FUNCTION_BLOCK TM3BC_Ethe_yYhtt9jWKUOJs (* Composite Function Block Type *)
  (* Standard: 61499-2 *)
  (* Version 0.0, 4/12/2022, Schneider Electric, template *)
  PACKAGE Main;
  {SET_ATTRIBUTE(Signature, 9B-51-86-C6-44-F1-B9-23-4E-CE-E4-D3-BB-FD-BE-0A-D2-5B-5E-A3-24-21-0B-6D-81-3C-00-8F-1B-F1-B9-BB-43-CA-DC-29-26-A0-D3-07-47-84-6D-56-70-09-2E-2C-30-58-B0-D9-37-4B-26-3D-BF-E3-73-7B-3A-E4-6A-55_67-4B-EE-2B-F7-15-C2-07-6B-CD-FB-3F-4A-FB-6C-FA-FE-85-84-91-EA-8A-10-A4-3E-5F-A5-D7-87-43-15-4E-8E-61-10-AD-23-0C-80-F7-8B-ED-9D-C9-E2-50-D4-40-3E-AD-16-B1-1E-C7-18-6C-9F-7C-EF-80-0E-8A-1D-44)}
  {SET_ATTRIBUTE(CreationMethod, Generic)}
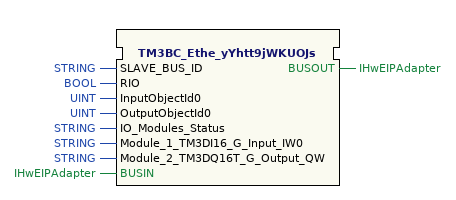
  VAR_INPUT
    SLAVE_BUS_ID : STRING; {SET_ATTRIBUTE(Configuration.HWConfiguration.HideInHwConfigurator, False)} {SET_ATTRIBUTE(Configuration.HWConfiguration.InheritInstanceName, True)}
    RIO : BOOL; {SET_ATTRIBUTE(Configuration.HWConfiguration.HideInHwConfigurator, True)} {SET_ATTRIBUTE(Configuration.HWConfiguration.ReadOnlyInHwConfigurator, True)}
    InputObjectId0 : UINT; (* Object ID of Input connection 0 *) {SET_ATTRIBUTE(Configuration.HWConfiguration.ReadOnlyInHwConfigurator, True)}
    OutputObjectId0 : UINT; (* Object ID of Output connection 0 *) {SET_ATTRIBUTE(Configuration.HWConfiguration.ReadOnlyInHwConfigurator, True)}
    IO_Modules_Status : STRING;
    Module_1_TM3DI16_G_Input_IW0 : STRING;
    Module_2_TM3DQ16T_G_Output_QW : STRING;
  END_VAR
  SOCKETS
    BUSIN : IHwEIPAdapter;
  END_SOCKETS
  PLUGS
    BUSOUT : IHwEIPAdapter;
  END_PLUGS
  FBS
    CONFIG : TEMPLATE_CONFIGURATION(ConnectionCount := 1);
    GetInstanceName : GET_INSTANCE_NAME(instanceLevel := 1);
    LogicalAndConnectionHealth : AND_88A3DD8EC65DD11C(IN2 := TRUE); {SET_ATTRIBUTE(Configuration.GenericFBType.InterfaceParams, Runtime.Standard#CNT:=2;OUT:BOOL)}
    fp : BaseFaceplate;
    busout_Connection_Check : CONNECTION_TEST(IOName := 'BUSOUT');
    SwitchConnectionCheck : E_SWITCH;
    SelectLastSlotNo : DS_SELECTX_29841900CAFD143A; {SET_ATTRIBUTE(Configuration.GenericFBType.InterfaceParams, Runtime.Standard#CNTX:=2;CNTY:=1;DI${CNTX,_,CNTY$}:UDINT)}
    SelectHealthAdapters : DS_SELECTX_2536758B411A6CE51; {SET_ATTRIBUTE(Configuration.GenericFBType.InterfaceParams, Runtime.Standard#CNTX:=2;CNTY:=1;DI${CNTX,_,CNTY$}:BOOL)}
    SelectConnectionsConfig : DS_SELECTX_170BB6FE986585D03; {SET_ATTRIBUTE(Configuration.GenericFBType.InterfaceParams, Runtime.Standard#CNTX:=2;CNTY:=1;DI${CNTX,_,CNTY$}:Standard.IoEtherNetIP.ConfigurationAC)}
    NOBUSCOUPLER : NOT_42C76073DCEB1A7A; {SET_ATTRIBUTE(Configuration.GenericFBType.InterfaceParams, Runtime.Standard#CNT:=1;OUT${CNT$}:BOOL)}
    CONNECTION0 : TEMPLATE_BUS_DEVICE_SLOT_NO(ConnectionIndex := 0);
    EIPConnectionInput0 : BUSDEVICE(QI := TRUE, ISBITDEVICE := FALSE, NINPUTBITS := 48);
    EIPConnectionOutput0 : BUSDEVICE(QI := TRUE, ISBITDEVICE := FALSE, NOUTPUTBITS := 16);
    ConfigConnection0 : AdapterSpecificCommon(connectionName := 'Connection_0', adapterIP := '', inputSize := 48, outputSize := 16);
    Event_OC_read_0_0 : EVENTCHAIN(NAME := 'EIP_HW_OC_INIT', PRIO := 1, TIMEOUT := T#10ms, DELAY := T#0ms);
    ioDataIn_0_0 : templateItemInputUDINT(Offset := 0, PdAnyInQI := TRUE, ForceValue := FALSE);
    Event_OC_read_0_1 : EVENTCHAIN(NAME := 'EIP_HW_OC_INIT', PRIO := 1, TIMEOUT := T#10ms, DELAY := T#0ms);
    ioDataIn_0_1 : templateItemInputWORD(Offset := 32, PdAnyInQI := TRUE, ForceValue := FALSE);
    Event_OC_write_0_2 : EVENTCHAIN(NAME := 'EIP_HW_OC_INIT', PRIO := 1, TIMEOUT := T#10ms, DELAY := T#0ms);
    ioDataOut_0_2 : templateItemOutputWORD(Offset := 0, PdAnyOutQI := TRUE);
  END_FBS
  EVENT_CONNECTIONS
    LogicalAndConnectionHealth.CNF TO fp.REQ_CHILDREN;
    fp.INITO TO busout_Connection_Check.REQ;
    CONFIG.INITO TO GetInstanceName.REQ;
    BUSOUT.INITO TO SelectLastSlotNo.REQ1;
    SelectLastSlotNo.IND TO BUSIN.INITO;
    busout_Connection_Check.E_NOT_CONNECTED TO SelectLastSlotNo.REQ2;
    busout_Connection_Check.E_CONNECTED TO BUSOUT.INIT;
    BUSOUT.HEALTHADAPTERS_RAISE TO SelectHealthAdapters.REQ1;
    SelectHealthAdapters.IND TO BUSIN.HEALTHADAPTERS_RAISE;
    BUSIN.INIT TO NOBUSCOUPLER.REQ;
    NOBUSCOUPLER.CNF TO CONFIG.INIT;
    SwitchConnectionCheck.EO0 TO SelectHealthAdapters.REQ2;
    SwitchConnectionCheck.EO1 TO BUSOUT.RECEIVE_HEALTHADAPTERS;
    BUSOUT.CONFIG_RAISE TO SelectConnectionsConfig.REQ1;
    SelectConnectionsConfig.IND TO BUSIN.CONFIG_RAISE;
    CONNECTION0.INITO TO EIPConnectionInput0.INIT;
    GetInstanceName.CNF TO CONNECTION0.INIT;
    BUSIN.RECEIVE_HEALTHADAPTERS TO ConfigConnection0.CONNECTION_HEALTH_RECEIVE_PREVIOUS_HEALTH;
    ConfigConnection0.HEALTH_CONNECTIONS_IND TO SwitchConnectionCheck.EI;
    ConfigConnection0.INITO TO fp.INIT;
    EIPConnectionInput0.INITO TO EIPConnectionOutput0.INIT;
    EIPConnectionOutput0.INITO TO ConfigConnection0.INIT;
    ConfigConnection0.HEALTH_IND TO LogicalAndConnectionHealth.REQ;
    ConfigConnection0.INITO TO SelectConnectionsConfig.REQ2;
    ConfigConnection0.INITO TO ioDataIn_0_0.INIT;
    ConfigConnection0.HEALTH_IND_INPUT TO ioDataIn_0_0.HEALTH_UPDATE_REQ;
    Event_OC_read_0_0.EO TO Event_OC_read_0_0.ACK;
    Event_OC_read_0_0.EO TO ioDataIn_0_0.OC_REQ;
    ConfigConnection0.INITO TO ioDataIn_0_1.INIT;
    ConfigConnection0.HEALTH_IND_INPUT TO ioDataIn_0_1.HEALTH_UPDATE_REQ;
    Event_OC_read_0_1.EO TO Event_OC_read_0_1.ACK;
    Event_OC_read_0_1.EO TO ioDataIn_0_1.OC_REQ;
    ConfigConnection0.INITO TO ioDataOut_0_2.INIT;
    ConfigConnection0.HEALTH_IND_OUTPUT TO ioDataOut_0_2.HEALTH_UPDATE_REQ;
    Event_OC_write_0_2.EO TO Event_OC_write_0_2.ACK;
    Event_OC_write_0_2.EO TO ioDataOut_0_2.OC_REQ;
  END_CONNECTIONS
  DATA_CONNECTIONS
    LogicalAndConnectionHealth.OUT TO fp.childrenHealth;
    GetInstanceName.instanceName TO fp.instanceName;
    BUSIN.busId TO BUSOUT.busId;
    BUSIN.diagBusId TO BUSOUT.diagBusId;
    BUSOUT.healthAdapters_Raise TO SelectHealthAdapters.DI1_1;
    SelectHealthAdapters.OUT1 TO BUSIN.healthAdapters_Raise;
    busout_Connection_Check.Connected TO SwitchConnectionCheck.G;
    BUSOUT.config_Raise TO SelectConnectionsConfig.DI1_1;
    SelectConnectionsConfig.OUT1 TO BUSIN.config_Raise;
    CONFIG.NextSlotNo TO BUSOUT.nextSlotNo;
    BUSIN.busId TO CONFIG.BusId;
    SLAVE_BUS_ID TO CONFIG.SlaveBusId;
    BUSIN.nextSlotNo TO CONFIG.SlotNo;
    RIO TO NOBUSCOUPLER.IN1;
    NOBUSCOUPLER.OUT1 TO CONFIG.NeedsBusCoupler;
    BUSIN.diagHealthSlotNo TO BUSOUT.diagHealthSlotNo;
    SelectLastSlotNo.OUT1 TO BUSIN.lastSlotNo;
    BUSOUT.lastSlotNo TO SelectLastSlotNo.DI1_1;
    CONFIG.LastSlotNoUsed TO SelectLastSlotNo.DI2_1;
    CONFIG.BusCouplerBusId TO EIPConnectionInput0.BUS_ID;
    CONFIG.BusCouplerBusId TO EIPConnectionOutput0.BUS_ID;
    CONNECTION0.ConnectionSlotInput TO ConfigConnection0.adapterSlot;
    CONNECTION0.ConnectionSlotInput TO EIPConnectionInput0.SLOT_NO;
    CONNECTION0.ConnectionSlotOutput TO EIPConnectionOutput0.SLOT_NO;
    CONFIG.FirstBusDeviceSlotInput TO CONNECTION0.FirstSlot;
    ConfigConnection0.configAC TO SelectConnectionsConfig.DI2_1;
    GetInstanceName.instanceName TO ConfigConnection0.adapterName;
    BUSIN.diagBusId TO ConfigConnection0.diagBusId;
    BUSIN.diagHealthSlotNo TO ConfigConnection0.diagHealthSlotNo;
    ConfigConnection0.health TO LogicalAndConnectionHealth.IN1;
    BUSIN.healthAdapters TO ConfigConnection0.healthConnectionsIn;
    ConfigConnection0.healthConnectionsOut TO SelectHealthAdapters.DI2_1;
    ConfigConnection0.healthConnectionsOut TO BUSOUT.healthAdapters;
    CONFIG.BusCouplerBusId TO ioDataIn_0_0.BusId;
    CONNECTION0.ConnectionSlotInput TO ioDataIn_0_0.SlotNo;
    ConfigConnection0.healthInput TO ioDataIn_0_0.HealthBit;
    IO_Modules_Status TO ioDataIn_0_0.SymLinkName;
    CONFIG.BusCouplerBusId TO ioDataIn_0_1.BusId;
    CONNECTION0.ConnectionSlotInput TO ioDataIn_0_1.SlotNo;
    ConfigConnection0.healthInput TO ioDataIn_0_1.HealthBit;
    Module_1_TM3DI16_G_Input_IW0 TO ioDataIn_0_1.SymLinkName;
    CONFIG.BusCouplerBusId TO ioDataOut_0_2.BusId;
    CONNECTION0.ConnectionSlotOutput TO ioDataOut_0_2.SlotNo;
    ConfigConnection0.healthOutput TO ioDataOut_0_2.HealthBit;
    Module_2_TM3DQ16T_G_Output_QW TO ioDataOut_0_2.SymLinkName;
    InputObjectId0 TO ConfigConnection0.inputObjectId;
    OutputObjectId0 TO ConfigConnection0.outputObjectId;
  END_CONNECTIONS
END_FUNCTION_BLOCK
